// TIA Portal V19 export
VAR_GLOBAL   // PLC tag table "JB_IO"
   JB_CutHead_Ls_Rest AT %I130.0 : Bool;   // 882SQ1
   JB_CutHead_Ls_Work AT %I130.1 : Bool;   // 882SQ2
   JB_PinchR_V_Close AT %Q132.0 : Bool;   // 904YV2
   JB_PinchR_Ls_Open AT %I130.4 : Bool;   // 904SQ1
   JB_PinchR_V_Open AT %Q131.7 : Bool;   // 904YV1
   JB_ClampEntry_Ls_Open AT %I130.2 : Bool;   // 883SQ1
   JB_ClampEntry_V_Work AT %Q131.4 : Bool;   // 883YV2
   JB_ClampEntry_V_Rest AT %Q131.3 : Bool;   // 883YV1
   JB_ClampExit_Ls_Rest AT %I130.3 : Bool;   // 884SQ1
   JB_ClampExit_V_Work AT %Q131.6 : Bool;   // 884YV2
   JB_ClampExit_V_Rest AT %Q131.5 : Bool;   // 884YV1
   JB_AI_Torch_Speed_Potentiometer AT %IW900 : Int;   // 463A1 - 328RP1
   JB_V_Libera_Apre AT %Q132.1 : Bool;   // 906
   JB_V_Libera_Chiude AT %Q132.2 : Bool;   // 906
   Controllo_Spessore_Lamiera_V_Soffio_Pulizia AT %Q131.2 : Bool;   // 870YV1
   JB_Welder_K_ON AT %Q123.0 : Bool;   // 880KA1
   JB_AspiratoreBanco_FbkRun AT %I143.4 : Bool;
   JB_AspiratoreBanco_KmRun AT %Q123.1 : Bool;   // 881KA1
END_VAR
